(* IEC 61131-3 sources: test/Class/SfcClass_Step0, 1 file *)

(* ---- SfcClass_Step0.st ---- *)
(*!
<Class
	Name               = "SfcClass_Step0"
	Revision           = "0.0"
	RealtimeTask       = "false"
	CyclicTask         = "false"
	BackgroundTask     = "false"
	Sigmatek           = "false"
	OSInterface        = "false"
	HighPriority       = "false"
	Automatic          = "false"
	UpdateMode         = "Prescan"
	SharedCommandTable = "true"
	Objectsize         = "(284,120)">
	<Channels>
	</Channels>
	<Network Name="SfcClass_Step0">
		<!-- List of Components in this network -->
		<Components>
			<Object
				Name       = "_base"
				Class      = "Sfc_Step_Base"
				Position   = "(218,120)"
				Visualized = "true"
				Remotely   = "true">
				<Channels>
					<Server Name="Itf"/>
					<Server Name="T"/>
					<Server Name="X"/>
					<Client Name="CallTransition"/>
					<Client Name="LogonToInvoker"/>
				</Channels>
			</Object>
		</Components>
		<Comments>
		</Comments>
		<!-- List of Connections in this network -->
		<Connections>
			<Connection Source="this.Itf" Destination="_base.Itf" Vertices="(690,210),(518,210),"/>
			<Connection Source="this.X" Destination="_base.X" Vertices="(690,270),(518,270),"/>
			<Connection Source="this.T" Destination="_base.T" Vertices="(690,330),(518,330),"/>
			<Connection Source="_base.LogonToInvoker" Destination="this.LogonToInvoker" Vertices="(230,210),(38,210),"/>
			<Connection Source="_base.CallTransition" Destination="this.CallTransition" Vertices="(230,270),(38,270),"/>
		</Connections>
		<!-- Headerfiles -->
		<Options>
		</Options>
	</Network>
</Class>
*)
#pragma using Sfc_Step_Base

SfcClass_Step0 : CLASS
: Sfc_Step_Base
  //Servers:
  //Clients:
  //Variables:
  //Functions:
				//! <Function Name="OnActive" Hidden="true"/>
	FUNCTION VIRTUAL OnActive;
				//! <Function Name="OnInactive" Hidden="true"/>
	FUNCTION VIRTUAL OnInactive;
  //Tables:
	FUNCTION @STD
		VAR_OUTPUT
			ret_code	: CONFSTATES;
		END_VAR;
	FUNCTION GLOBAL TAB @CT_;
END_CLASS;

FUNCTION VIRTUAL SfcClass_Step0::OnActive

END_FUNCTION
FUNCTION VIRTUAL SfcClass_Step0::OnInactive

END_FUNCTION
